// Mitsubishi GX Works2 project: pneumatic_control_2   PLC: Q03UDV

PROGRAM MAIN
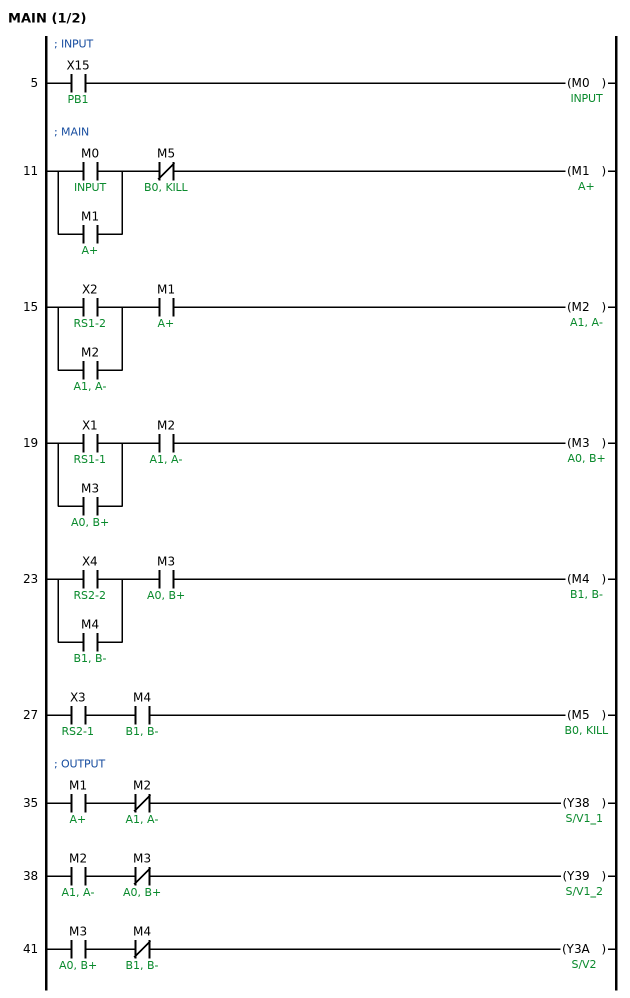
; INPUT
5     LD      X15  ; PB1
      OUT     M0  ; INPUT
; MAIN
11    LD      M0  ; INPUT
      OR      M1  ; A+
      ANI     M5  ; B0, KILL
      OUT     M1  ; A+
15    LD      X2  ; RS1-2
      OR      M2  ; A1, A-
      AND     M1  ; A+
      OUT     M2  ; A1, A-
19    LD      X1  ; RS1-1
      OR      M3  ; A0, B+
      AND     M2  ; A1, A-
      OUT     M3  ; A0, B+
23    LD      X4  ; RS2-2
      OR      M4  ; B1, B-
      AND     M3  ; A0, B+
      OUT     M4  ; B1, B-
27    LD      X3  ; RS2-1
      AND     M4  ; B1, B-
      OUT     M5  ; B0, KILL
; OUTPUT
35    LD      M1  ; A+
      ANI     M2  ; A1, A-
      OUT     Y38  ; S/V1_1
38    LD      M2  ; A1, A-
      ANI     M3  ; A0, B+
      OUT     Y39  ; S/V1_2
41    LD      M3  ; A0, B+
      ANI     M4  ; B1, B-
      OUT     Y3A  ; S/V2
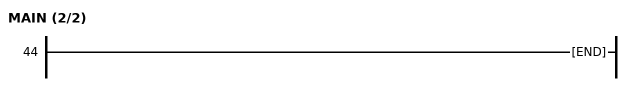
44    END
END_PROGRAM
